// TIA Portal V19 export
DATA_BLOCK "LEVEL BUFF"   // DB14
{ S7_Optimized_Access := 'TRUE' }
// stored: MemoryReserve 100
   VAR RETAIN
      "SYRUP MFG_TEMP" : Int;
      "SYRUP MFG_COOLING" : Int;
      "SYRUP MFG_VACCUM" : Int;
      "SYRUP MFG_LOAD CELL" : Int;
      PREMIXING_TEMP : Int;
      PREMIXING_COOLING : Int;
      PREMIXING_VACCUM : Int;
      "PREMIXING_LOAD CELL" : Int;
      SUGAR_TEMP : Int;
      SUGAR_VACCUM : Int;
      "SUGAR_LOAD CELL" : Int;
   END_VAR
   VAR
      AUTO : Struct
         "MFG LOAD CELL" : Int;
         "MFG TEMP MIN_MAX BUFF" : Int;
         "MFG VACUUM MIN_MAX BUFF" : Int;
         "PREMIXING LOAD CELL" : Int;
         "PREMIXING TEMP MIN_MAX BUFF" : Int;
         "PREMIXING VACUUM MIN_MAX BUFF" : Int;
         "SUGAR LOAD CELL" : Int;
         "SUGAR TEMP MIN_MAX BUFF" : Int;
         "SUGAR VACUUM MIN_MAX BUFF" : Int;
      END_STRUCT;
   END_VAR
BEGIN
END_DATA_BLOCK
